FUNCTION_BLOCK FB_DigitalInputSensor
VAR_INPUT
	on : BOOL;
	inTime : TIME;
	
END_VAR

VAR_OUTPUT
	digitalFiltered : BOOL;
END_VAR
VAR
	tOnGetTime : TON;
END_VAR

tOnGetTime(PT := inTime);
IF on THEN
	tOnGetTime.IN := TRUE;
	IF tOnGetTime.Q THEN
		digitalFiltered := TRUE;
	ELSE digitalFiltered := FALSE;
	END_IF
ELSE tOnGetTime.IN := FALSE;
END_IF

END_FUNCTION_BLOCK

(* stored: Version 1.1.0.1, ProductVersion 3.1.4024.14
   POU FB_DidigtalInputSensor: Id {a033c98f-67b5-4571-aca6-6455c4e13572}, SpecialFunc None *)
